SUBAPPLICATION Uebung_094a (* Beispiel für QI anstelle Permit *)
  (* Standard: 61499-2; Description: Copyright (c) 2023 Meisterschulen am Ostbahnhof This program and the accompanying materials are made available under the terms of the Eclipse Public License 2.0 which is available at https://www.eclipse.org/legal/epl-2.0/ SPDX-License-Identifier: EPL-2.0 Beispiel für E_CTD Aufwärts zählen UAO Curriculum Module 3 - The IEC 61499 Standard, Seite 93 *)
  (* Version 1.0, 2023-10-23, Franz Höpfinger, Meisterschulen am Ostbahnhof *)
  PACKAGE Uebungen;
  IMPORT logiBUS::io::DI::logiBUS_DI::Input_I1;
  IMPORT logiBUS::io::DI::logiBUS_DI::Input_I2;
  IMPORT logiBUS::io::DI::logiBUS_DI_Events::BUTTON_SINGLE_CLICK;
  IMPORT logiBUS::io::DQ::logiBUS_DO::Output_Q1;
  IMPORT logiBUS::io::DQ::logiBUS_DO::Output_Q2;
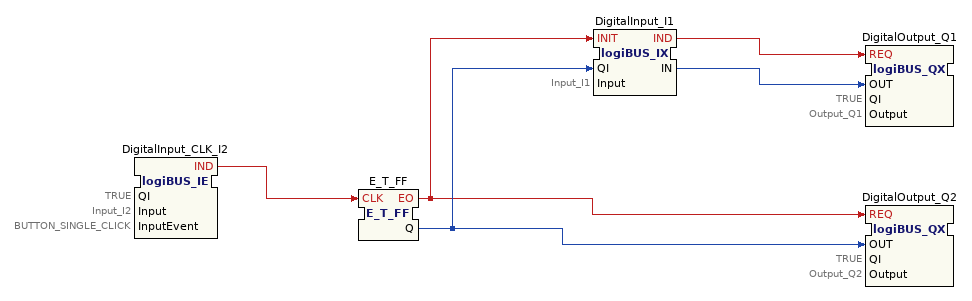
  FBS
    DigitalInput_I1 : logiBUS::io::DI::logiBUS_IX(Input := Input_I1);
    DigitalInput_CLK_I2 : logiBUS::io::DI::logiBUS_IE(QI := TRUE, Input := Input_I2, InputEvent := BUTTON_SINGLE_CLICK);
    E_T_FF : iec61499::events::E_T_FF;
    DigitalOutput_Q1 : logiBUS::io::DQ::logiBUS_QX(QI := TRUE, Output := Output_Q1);
    DigitalOutput_Q2 : logiBUS::io::DQ::logiBUS_QX(QI := TRUE, Output := Output_Q2);
  END_FBS
  EVENT_CONNECTIONS
    DigitalInput_CLK_I2.IND TO E_T_FF.CLK;
    DigitalInput_I1.IND TO DigitalOutput_Q1.REQ;
    E_T_FF.EO TO DigitalInput_I1.INIT;
    E_T_FF.EO TO DigitalOutput_Q2.REQ;
  END_CONNECTIONS
  DATA_CONNECTIONS
    DigitalInput_I1.IN TO DigitalOutput_Q1.OUT;
    E_T_FF.Q TO DigitalInput_I1.QI;
    E_T_FF.Q TO DigitalOutput_Q2.OUT;
  END_CONNECTIONS
END_SUBAPPLICATION
